// TIA Portal V19 export
FUNCTION "Valve Control" : Void   // FC5, LAD
{ S7_Optimized_Access := 'TRUE' }
// stored: SetENOAutomatically false
BEGIN

REGION Network 1: IBC Valve Control
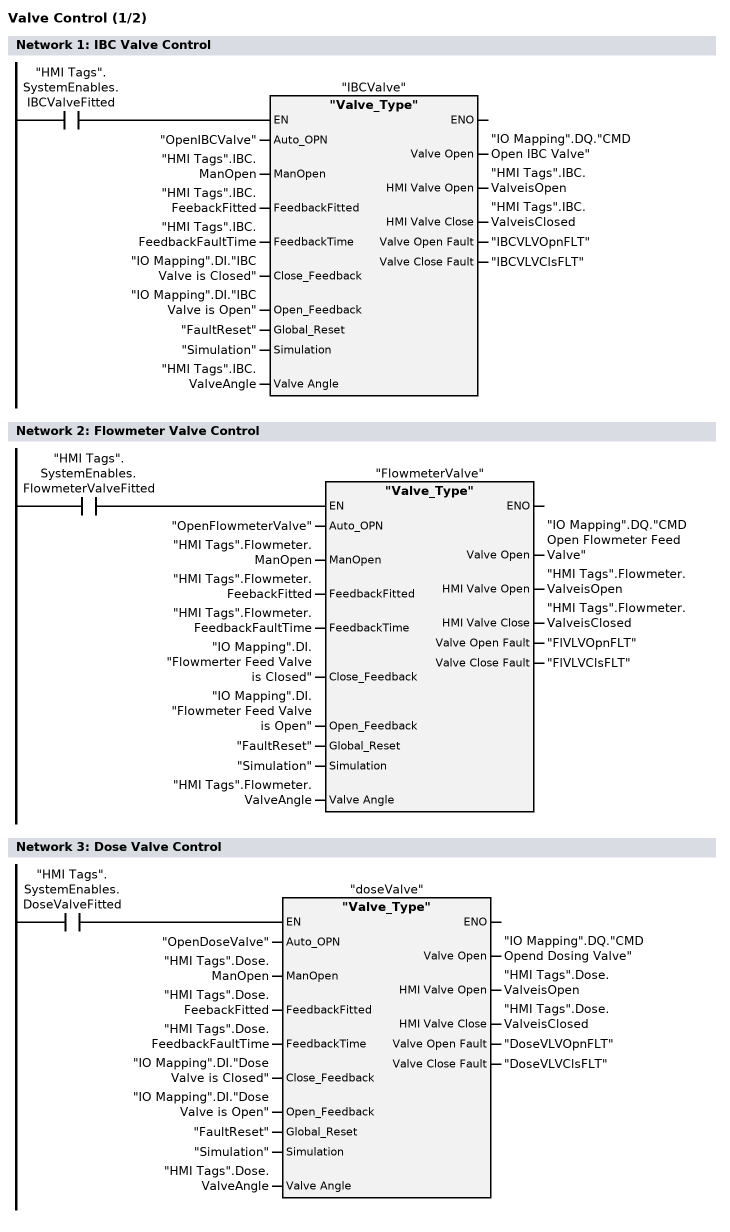
   RUNG wire#powerrail
      Contact( "HMI Tags".SystemEnables.IBCValveFitted )
      "IBCValve"(Auto_OPN := "OpenIBCValve", ManOpen := "HMI Tags".IBC.ManOpen, FeedbackFitted := "HMI Tags".IBC.FeebackFitted, FeedbackTime := "HMI Tags".IBC.FeedbackFaultTime, Close_Feedback := "IO Mapping".DI."IBC Valve is Closed", Open_Feedback := "IO Mapping".DI."IBC Valve is Open", Global_Reset := "FaultReset", Simulation := "Simulation", "Valve Angle" := "HMI Tags".IBC.ValveAngle, "Valve Open" => "IO Mapping".DQ."CMD Open IBC Valve", "HMI Valve Open" => "HMI Tags".IBC.ValveisOpen, "HMI Valve Close" => "HMI Tags".IBC.ValveisClosed, "Valve Open Fault" => "IBCVLVOpnFLT", "Valve Close Fault" => "IBCVLVClsFLT")
   END_RUNG
   // the same network as SCL:
   IF "HMI Tags".SystemEnables.IBCValveFitted THEN
       "IBCValve"(Auto_OPN := "OpenIBCValve",   // "Valve_Type"
                  ManOpen := "HMI Tags".IBC.ManOpen,
                  FeedbackFitted := "HMI Tags".IBC.FeebackFitted,
                  FeedbackTime := "HMI Tags".IBC.FeedbackFaultTime,
                  Close_Feedback := "IO Mapping".DI."IBC Valve is Closed",
                  Open_Feedback := "IO Mapping".DI."IBC Valve is Open",
                  Global_Reset := "FaultReset",
                  Simulation := "Simulation",
                  "Valve Angle" := "HMI Tags".IBC.ValveAngle,
                  "Valve Open" => "IO Mapping".DQ."CMD Open IBC Valve",
                  "HMI Valve Open" => "HMI Tags".IBC.ValveisOpen,
                  "HMI Valve Close" => "HMI Tags".IBC.ValveisClosed,
                  "Valve Open Fault" => "IBCVLVOpnFLT",
                  "Valve Close Fault" => "IBCVLVClsFLT");
   END_IF;
END_REGION

REGION Network 2: Flowmeter Valve Control
   RUNG wire#powerrail
      Contact( "HMI Tags".SystemEnables.FlowmeterValveFitted )
      "FlowmeterValve"(Auto_OPN := "OpenFlowmeterValve", ManOpen := "HMI Tags".Flowmeter.ManOpen, FeedbackFitted := "HMI Tags".Flowmeter.FeebackFitted, FeedbackTime := "HMI Tags".Flowmeter.FeedbackFaultTime, Close_Feedback := "IO Mapping".DI."Flowmerter Feed Valve is Closed", Open_Feedback := "IO Mapping".DI."Flowmeter Feed Valve is Open", Global_Reset := "FaultReset", Simulation := "Simulation", "Valve Angle" := "HMI Tags".Flowmeter.ValveAngle, "Valve Open" => "IO Mapping".DQ."CMD Open Flowmeter Feed Valve", "HMI Valve Open" => "HMI Tags".Flowmeter.ValveisOpen, "HMI Valve Close" => "HMI Tags".Flowmeter.ValveisClosed, "Valve Open Fault" => "FlVLVOpnFLT", "Valve Close Fault" => "FlVLVClsFLT")
   END_RUNG
   // the same network as SCL:
   IF "HMI Tags".SystemEnables.FlowmeterValveFitted THEN
       "FlowmeterValve"(Auto_OPN := "OpenFlowmeterValve",   // "Valve_Type"
                        ManOpen := "HMI Tags".Flowmeter.ManOpen,
                        FeedbackFitted := "HMI Tags".Flowmeter.FeebackFitted,
                        FeedbackTime := "HMI Tags".Flowmeter.FeedbackFaultTime,
                        Close_Feedback := "IO Mapping".DI."Flowmerter Feed Valve is Closed",
                        Open_Feedback := "IO Mapping".DI."Flowmeter Feed Valve is Open",
                        Global_Reset := "FaultReset",
                        Simulation := "Simulation",
                        "Valve Angle" := "HMI Tags".Flowmeter.ValveAngle,
                        "Valve Open" => "IO Mapping".DQ."CMD Open Flowmeter Feed Valve",
                        "HMI Valve Open" => "HMI Tags".Flowmeter.ValveisOpen,
                        "HMI Valve Close" => "HMI Tags".Flowmeter.ValveisClosed,
                        "Valve Open Fault" => "FlVLVOpnFLT",
                        "Valve Close Fault" => "FlVLVClsFLT");
   END_IF;
END_REGION

REGION Network 3: Dose Valve Control
   RUNG wire#powerrail
      Contact( "HMI Tags".SystemEnables.DoseValveFitted )
      "doseValve"(Auto_OPN := "OpenDoseValve", ManOpen := "HMI Tags".Dose.ManOpen, FeedbackFitted := "HMI Tags".Dose.FeebackFitted, FeedbackTime := "HMI Tags".Dose.FeedbackFaultTime, Close_Feedback := "IO Mapping".DI."Dose Valve is Closed", Open_Feedback := "IO Mapping".DI."Dose Valve is Open", Global_Reset := "FaultReset", Simulation := "Simulation", "Valve Angle" := "HMI Tags".Dose.ValveAngle, "Valve Open" => "IO Mapping".DQ."CMD Opend Dosing Valve", "HMI Valve Open" => "HMI Tags".Dose.ValveisOpen, "HMI Valve Close" => "HMI Tags".Dose.ValveisClosed, "Valve Open Fault" => "DoseVLVOpnFLT", "Valve Close Fault" => "DoseVLVClsFLT")
   END_RUNG
   // the same network as SCL:
   IF "HMI Tags".SystemEnables.DoseValveFitted THEN
       "doseValve"(Auto_OPN := "OpenDoseValve",   // "Valve_Type"
                   ManOpen := "HMI Tags".Dose.ManOpen,
                   FeedbackFitted := "HMI Tags".Dose.FeebackFitted,
                   FeedbackTime := "HMI Tags".Dose.FeedbackFaultTime,
                   Close_Feedback := "IO Mapping".DI."Dose Valve is Closed",
                   Open_Feedback := "IO Mapping".DI."Dose Valve is Open",
                   Global_Reset := "FaultReset",
                   Simulation := "Simulation",
                   "Valve Angle" := "HMI Tags".Dose.ValveAngle,
                   "Valve Open" => "IO Mapping".DQ."CMD Opend Dosing Valve",
                   "HMI Valve Open" => "HMI Tags".Dose.ValveisOpen,
                   "HMI Valve Close" => "HMI Tags".Dose.ValveisClosed,
                   "Valve Open Fault" => "DoseVLVOpnFLT",
                   "Valve Close Fault" => "DoseVLVClsFLT");
   END_IF;
END_REGION

REGION Network 4: Pump Valve Control
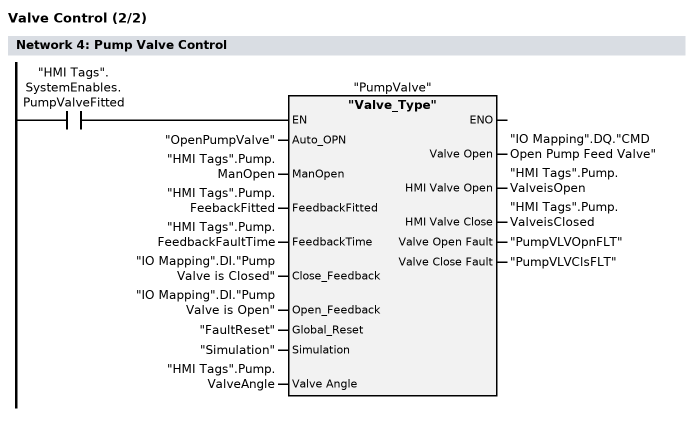
   RUNG wire#powerrail
      Contact( "HMI Tags".SystemEnables.PumpValveFitted )
      "PumpValve"(Auto_OPN := "OpenPumpValve", ManOpen := "HMI Tags".Pump.ManOpen, FeedbackFitted := "HMI Tags".Pump.FeebackFitted, FeedbackTime := "HMI Tags".Pump.FeedbackFaultTime, Close_Feedback := "IO Mapping".DI."Pump Valve is Closed", Open_Feedback := "IO Mapping".DI."Pump Valve is Open", Global_Reset := "FaultReset", Simulation := "Simulation", "Valve Angle" := "HMI Tags".Pump.ValveAngle, "Valve Open" => "IO Mapping".DQ."CMD Open Pump Feed Valve", "HMI Valve Open" => "HMI Tags".Pump.ValveisOpen, "HMI Valve Close" => "HMI Tags".Pump.ValveisClosed, "Valve Open Fault" => "PumpVLVOpnFLT", "Valve Close Fault" => "PumpVLVClsFLT")
   END_RUNG
   // the same network as SCL:
   IF "HMI Tags".SystemEnables.PumpValveFitted THEN
       "PumpValve"(Auto_OPN := "OpenPumpValve",   // "Valve_Type"
                   ManOpen := "HMI Tags".Pump.ManOpen,
                   FeedbackFitted := "HMI Tags".Pump.FeebackFitted,
                   FeedbackTime := "HMI Tags".Pump.FeedbackFaultTime,
                   Close_Feedback := "IO Mapping".DI."Pump Valve is Closed",
                   Open_Feedback := "IO Mapping".DI."Pump Valve is Open",
                   Global_Reset := "FaultReset",
                   Simulation := "Simulation",
                   "Valve Angle" := "HMI Tags".Pump.ValveAngle,
                   "Valve Open" => "IO Mapping".DQ."CMD Open Pump Feed Valve",
                   "HMI Valve Open" => "HMI Tags".Pump.ValveisOpen,
                   "HMI Valve Close" => "HMI Tags".Pump.ValveisClosed,
                   "Valve Open Fault" => "PumpVLVOpnFLT",
                   "Valve Close Fault" => "PumpVLVClsFLT");
   END_IF;
END_REGION
END_FUNCTION
